TYPE ST_Motor :
STRUCT
	Up,
	Down,
	Slow ,
	Brake :BOOL;
END_STRUCT
END_TYPE

(* stored: Version 1.1.0.1, ProductVersion 3.1.4024.11
   DUT ST_Motor: Id {49701605-1ef5-465f-8a2d-70cc7fc317e1} *)
